{attribute addProperty BoxType "KL8001"}
{attribute addProperty Id "Channel_1Channel_64E042E300"}
{attribute addProperty CRC "2007703693"}
{attribute addProperty SizeInBites "0"}
{attribute addProperty SizeInBytes "0"}
TYPE KL8001_77AB208D :
STRUCT
	{attribute addProperty Name "Channel_1"}
	Channel_1 : Channel_64E042E3;
END_STRUCT
END_TYPE

(* stored: Version 1.2.0.0, ProductVersion 3.1.4024.9
   DUT KL8001_77AB208D: Id {7dd73396-0d67-48c8-b892-2018092c9238} *)
